// TIA Portal project "5 Run - 2 Stop (1T)" (V16)

(* hardware
DEVICE "S7-1200 station_1"  S7-1200 Station
   slot 0: "Rack_0"  S7-1200 Rack  Rack  V1.0
   slot 1: "PLC_1"  CPU 1212C AC/DC/Rly  6ES7 212-1BE40-0XB0  V4.0
*)

// ===== PLC "PLC_1"  CPU 1212C AC/DC/Rly =====

VAR_GLOBAL   // PLC tag table "Default tag table"
   "start1" AT %I0.2 : Bool;
   "K1" AT %Q0.0 : Bool;
   "stop1" AT %I0.4 : Bool;
   "k2" AT %Q0.1 : Bool;
   "start2" AT %I0.3 : Bool;
   "T1 tag" AT %M0.0 : Bool;
   "T2 tag" AT %M0.1 : Bool;
   "X" AT %M0.2 : Bool;
   "stop 2S" AT %M1.0 : Bool;
   "tag_2" AT %M1.1 : Bool;
   "K3" AT %Q0.2 : Bool;
   "C2 TAG" AT %M0.3 : Bool;
   "C1 TAG" AT %M2.3 : Bool;
END_VAR

// folder: System blocks/Program resources

DATA_BLOCK "C1"   // DB1
{ S7_Optimized_Access := 'TRUE' }
AUTHOR : Simatic
FAMILY : IEC
NAME : CNTR
VERSION : 1.0
// stored: InstanceOfName IEC_COUNTER
"IEC_COUNTER"
BEGIN
END_DATA_BLOCK

DATA_BLOCK "T1"   // DB2
{ S7_Optimized_Access := 'TRUE' }
AUTHOR : Simatic
FAMILY : IEC
NAME : IEC_TMR
VERSION : 1.0
// stored: InstanceOfName IEC_TIMER
"IEC_TIMER"
BEGIN
END_DATA_BLOCK

DATA_BLOCK "C2"   // DB4
{ S7_Optimized_Access := 'TRUE' }
AUTHOR : Simatic
FAMILY : IEC
NAME : CNTR
VERSION : 1.0
// stored: InstanceOfName IEC_COUNTER
"IEC_COUNTER"
BEGIN
END_DATA_BLOCK

// folder: (top level)

ORGANIZATION_BLOCK "Main"   // OB1, LAD, ProgramCycle
TITLE = "Main Program Sweep (Cycle)"
{ S7_Optimized_Access := 'TRUE' }
VERSION : 0.1
   VAR_INPUT
      Initial_Call : Bool;   // Initial call of this OB
      Remanence : Bool;   // =True, if remanent data are available
   END_VAR
BEGIN

REGION Network 1: start
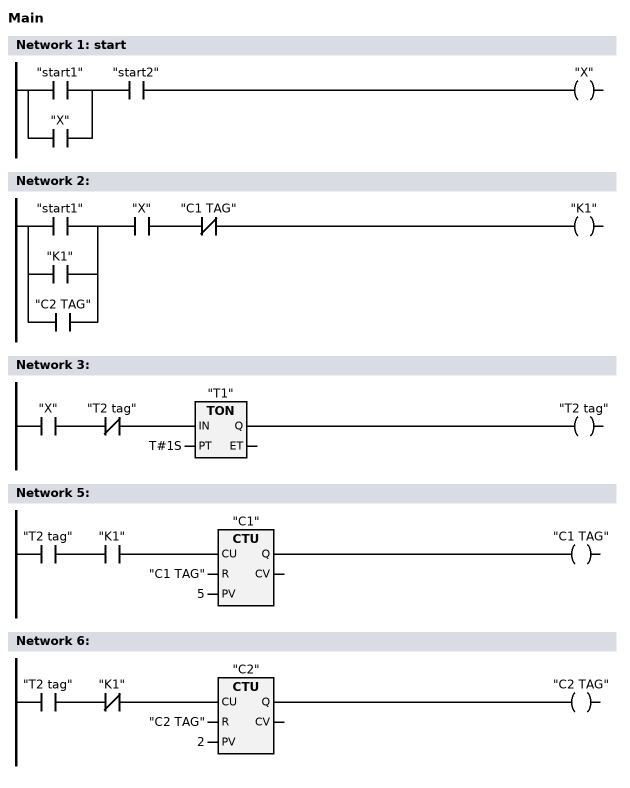
   RUNG wire#powerrail
      Contact( "start1" )
      wire#w1
      Contact( "start2" )
      Coil( "X" )
   END_RUNG
   RUNG wire#powerrail
      Contact( "X" )
   END_RUNG wire#w1
   // the same network as SCL:
   "X" := ("start1" OR "X") AND "start2";
END_REGION

REGION Network 2
   RUNG wire#powerrail
      Contact( "start1" )
      wire#w1
      Contact( "X" )
      I_Contact( "C1 TAG" )
      Coil( "K1" )
   END_RUNG
   RUNG wire#powerrail
      Contact( "K1" )
   END_RUNG wire#w1
   RUNG wire#powerrail
      Contact( "C2 TAG" )
   END_RUNG wire#w1
   // the same network as SCL:
   "K1" := ("start1" OR "K1" OR "C2 TAG") AND "X" AND NOT "C1 TAG";
END_REGION

REGION Network 3
   "T1".TON(IN := "X" AND NOT "T2 tag", PT := T#1S);
   "T2 tag" := "T1".Q;
END_REGION

REGION Network 5
   "C1".CTU(CU := "T2 tag" AND "K1", R := "C1 TAG", PV := 5);
   "C1 TAG" := "C1".Q;
END_REGION

REGION Network 6
   "C2".CTU(CU := "T2 tag" AND NOT "K1", R := "C2 TAG", PV := 2);
   "C2 TAG" := "C2".Q;
END_REGION
END_ORGANIZATION_BLOCK